// TIA Portal V18 export
FUNCTION_BLOCK "AndonMain"   // FB1, FBD
{ S7_Optimized_Access := 'TRUE' }
VERSION : 0.1
// stored: AutoNumber true, IsIECCheckEnabled false, IsRetainMemResEnabled false, MemoryReserve 100, SetENOAutomatically false, UDAEnableTagReadback false
   VAR
      fpBit_greenTrigger : Bool;
      AndonBoxASi_v2_Instance_8 { S7_SetPoint := 'True'} : "AndonBoxASi";
      AndonBoxASi_v2_Instance_9 { S7_SetPoint := 'True'} : "AndonBoxASi";
      AndonBoxASi_v2_Instance1 { S7_SetPoint := 'True'} : "AndonBoxASi";
      AndonBoxASi_v2_Instance2 { S7_SetPoint := 'True'} : "AndonBoxASi";
      AndonBoxASi_v2_Instance3 { S7_SetPoint := 'True'} : "AndonBoxASi";
      AndonBoxASi_v2_Instance4 { S7_SetPoint := 'True'} : "AndonBoxASi";
      AndonBoxASi_v2_Instance5 { S7_SetPoint := 'True'} : "AndonBoxASi";
      AndonBoxASi_v2_Instance6 { S7_SetPoint := 'True'} : "AndonBoxASi";
      AndonBoxASi_v2_Instance7 { S7_SetPoint := 'True'} : "AndonBoxASi";
      AndonBoxASi_v2_Instance10 { S7_SetPoint := 'True'} : "AndonBoxASi";
   END_VAR
   VAR_TEMP   // added for the SCL form of the ladder/FBD networks
      _w1 : Bool;
      _w2 : Bool;
   END_VAR
BEGIN

REGION Network 1: Green trigger
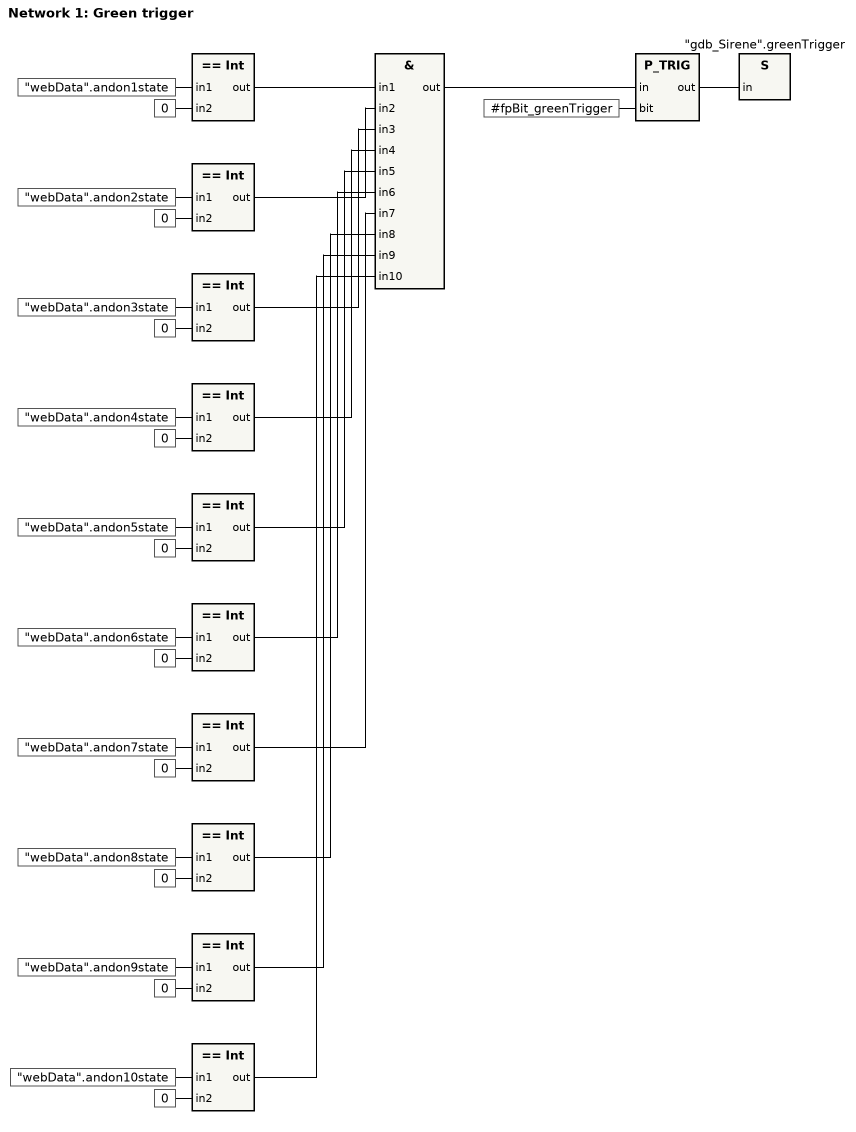
   #_w1 := ("webData".andon1state = 0) AND ("webData".andon2state = 0) AND ("webData".andon3state = 0) AND ("webData".andon4state = 0) AND ("webData".andon5state = 0) AND ("webData".andon6state = 0) AND ("webData".andon7state = 0) AND ("webData".andon8state = 0) AND ("webData".andon9state = 0) AND ("webData".andon10state = 0);
   #_w2 := #_w1 AND NOT #fpBit_greenTrigger;   // rising edge
   #fpBit_greenTrigger := #_w1;
   IF #_w2 THEN "gdb_Sirene".greenTrigger := TRUE; END_IF;
END_REGION

REGION Network 2: Andon1
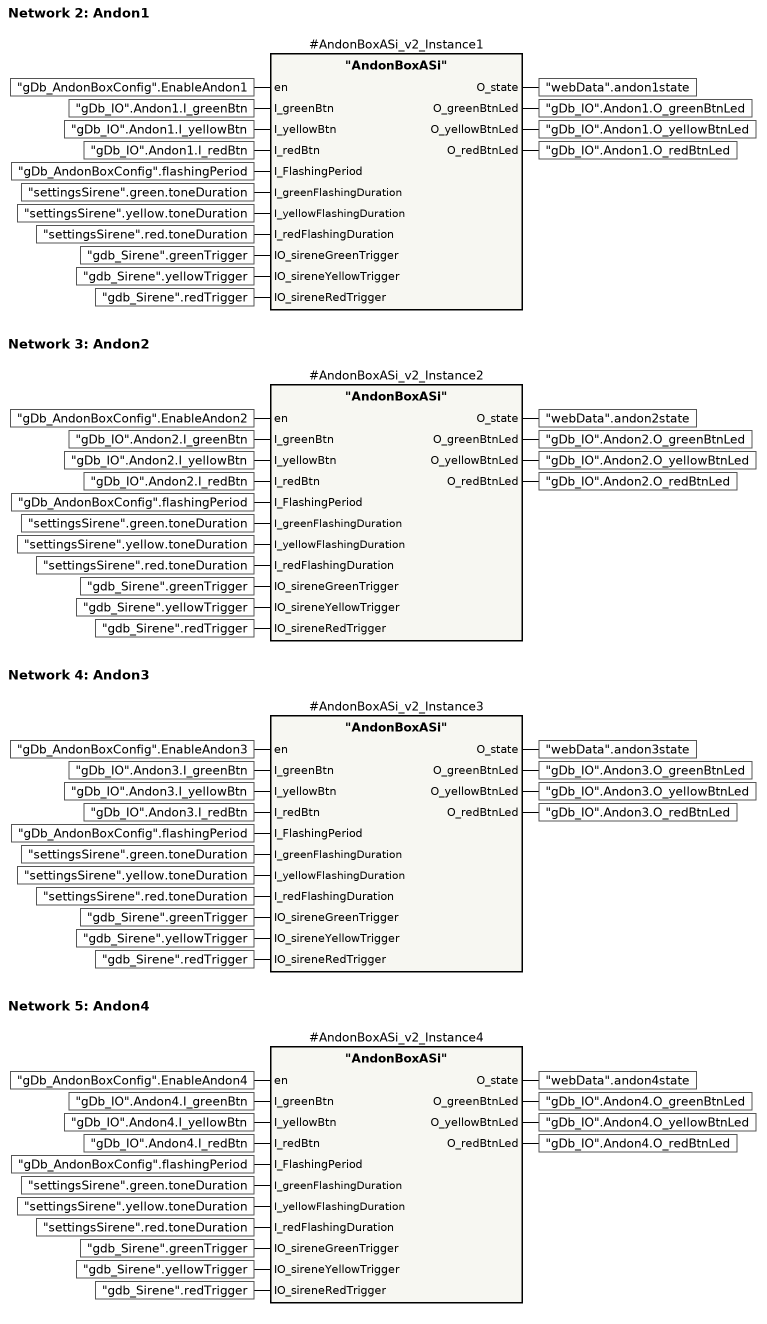
   IF "gDb_AndonBoxConfig".EnableAndon1 THEN
       #AndonBoxASi_v2_Instance1(I_greenBtn := "gDb_IO".Andon1.I_greenBtn,   // "AndonBoxASi"
                               I_yellowBtn := "gDb_IO".Andon1.I_yellowBtn,
                               I_redBtn := "gDb_IO".Andon1.I_redBtn,
                               I_FlashingPeriod := "gDb_AndonBoxConfig".flashingPeriod,
                               I_greenFlashingDuration := "settingsSirene".green.toneDuration,
                               I_yellowFlashingDuration := "settingsSirene".yellow.toneDuration,
                               I_redFlashingDuration := "settingsSirene".red.toneDuration,
                               IO_sireneGreenTrigger := "gdb_Sirene".greenTrigger,
                               IO_sireneYellowTrigger := "gdb_Sirene".yellowTrigger,
                               IO_sireneRedTrigger := "gdb_Sirene".redTrigger,
                               O_state => "webData".andon1state,
                               O_greenBtnLed => "gDb_IO".Andon1.O_greenBtnLed,
                               O_yellowBtnLed => "gDb_IO".Andon1.O_yellowBtnLed,
                               O_redBtnLed => "gDb_IO".Andon1.O_redBtnLed);
   END_IF;
END_REGION

REGION Network 3: Andon2
   IF "gDb_AndonBoxConfig".EnableAndon2 THEN
       #AndonBoxASi_v2_Instance2(I_greenBtn := "gDb_IO".Andon2.I_greenBtn,   // "AndonBoxASi"
                               I_yellowBtn := "gDb_IO".Andon2.I_yellowBtn,
                               I_redBtn := "gDb_IO".Andon2.I_redBtn,
                               I_FlashingPeriod := "gDb_AndonBoxConfig".flashingPeriod,
                               I_greenFlashingDuration := "settingsSirene".green.toneDuration,
                               I_yellowFlashingDuration := "settingsSirene".yellow.toneDuration,
                               I_redFlashingDuration := "settingsSirene".red.toneDuration,
                               IO_sireneGreenTrigger := "gdb_Sirene".greenTrigger,
                               IO_sireneYellowTrigger := "gdb_Sirene".yellowTrigger,
                               IO_sireneRedTrigger := "gdb_Sirene".redTrigger,
                               O_state => "webData".andon2state,
                               O_greenBtnLed => "gDb_IO".Andon2.O_greenBtnLed,
                               O_yellowBtnLed => "gDb_IO".Andon2.O_yellowBtnLed,
                               O_redBtnLed => "gDb_IO".Andon2.O_redBtnLed);
   END_IF;
END_REGION

REGION Network 4: Andon3
   IF "gDb_AndonBoxConfig".EnableAndon3 THEN
       #AndonBoxASi_v2_Instance3(I_greenBtn := "gDb_IO".Andon3.I_greenBtn,   // "AndonBoxASi"
                               I_yellowBtn := "gDb_IO".Andon3.I_yellowBtn,
                               I_redBtn := "gDb_IO".Andon3.I_redBtn,
                               I_FlashingPeriod := "gDb_AndonBoxConfig".flashingPeriod,
                               I_greenFlashingDuration := "settingsSirene".green.toneDuration,
                               I_yellowFlashingDuration := "settingsSirene".yellow.toneDuration,
                               I_redFlashingDuration := "settingsSirene".red.toneDuration,
                               IO_sireneGreenTrigger := "gdb_Sirene".greenTrigger,
                               IO_sireneYellowTrigger := "gdb_Sirene".yellowTrigger,
                               IO_sireneRedTrigger := "gdb_Sirene".redTrigger,
                               O_state => "webData".andon3state,
                               O_greenBtnLed => "gDb_IO".Andon3.O_greenBtnLed,
                               O_yellowBtnLed => "gDb_IO".Andon3.O_yellowBtnLed,
                               O_redBtnLed => "gDb_IO".Andon3.O_redBtnLed);
   END_IF;
END_REGION

REGION Network 5: Andon4
   IF "gDb_AndonBoxConfig".EnableAndon4 THEN
       #AndonBoxASi_v2_Instance4(I_greenBtn := "gDb_IO".Andon4.I_greenBtn,   // "AndonBoxASi"
                               I_yellowBtn := "gDb_IO".Andon4.I_yellowBtn,
                               I_redBtn := "gDb_IO".Andon4.I_redBtn,
                               I_FlashingPeriod := "gDb_AndonBoxConfig".flashingPeriod,
                               I_greenFlashingDuration := "settingsSirene".green.toneDuration,
                               I_yellowFlashingDuration := "settingsSirene".yellow.toneDuration,
                               I_redFlashingDuration := "settingsSirene".red.toneDuration,
                               IO_sireneGreenTrigger := "gdb_Sirene".greenTrigger,
                               IO_sireneYellowTrigger := "gdb_Sirene".yellowTrigger,
                               IO_sireneRedTrigger := "gdb_Sirene".redTrigger,
                               O_state => "webData".andon4state,
                               O_greenBtnLed => "gDb_IO".Andon4.O_greenBtnLed,
                               O_yellowBtnLed => "gDb_IO".Andon4.O_yellowBtnLed,
                               O_redBtnLed => "gDb_IO".Andon4.O_redBtnLed);
   END_IF;
END_REGION

REGION Network 6: Andon5
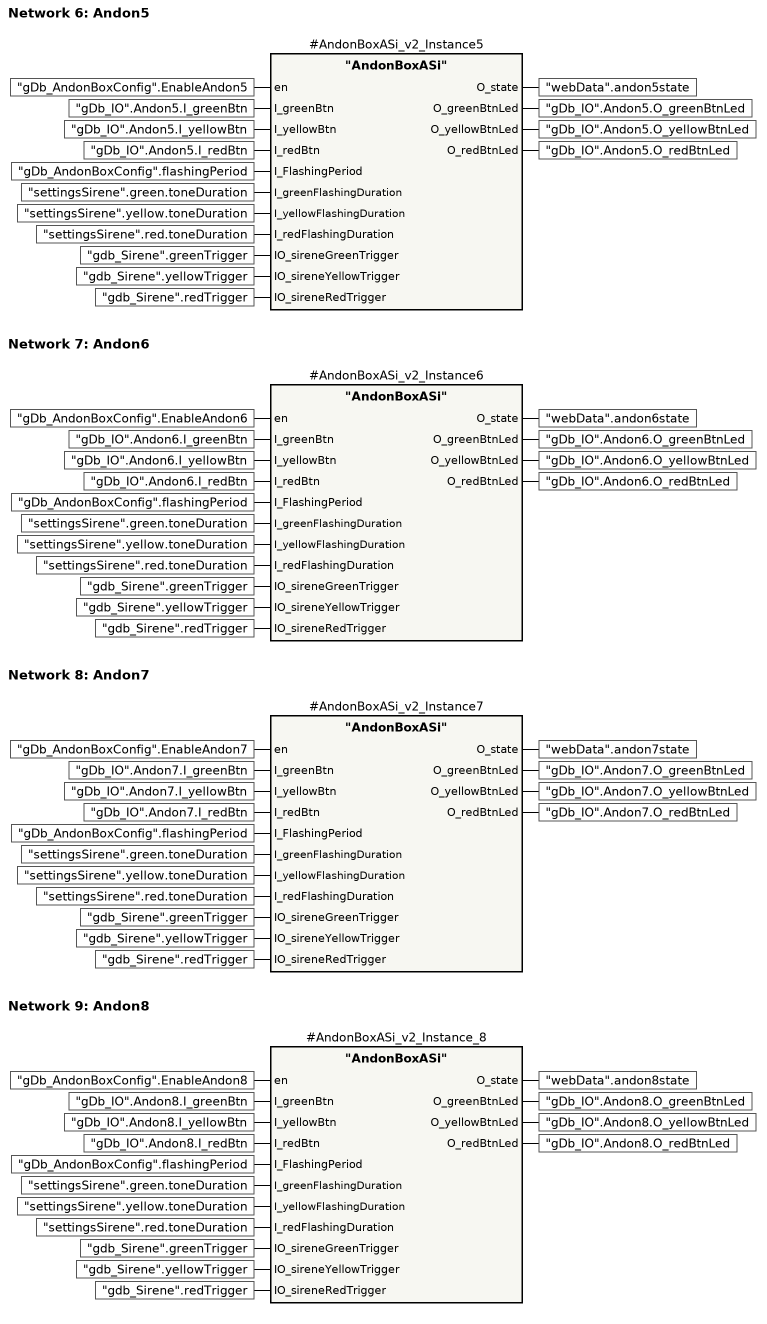
   IF "gDb_AndonBoxConfig".EnableAndon5 THEN
       #AndonBoxASi_v2_Instance5(I_greenBtn := "gDb_IO".Andon5.I_greenBtn,   // "AndonBoxASi"
                               I_yellowBtn := "gDb_IO".Andon5.I_yellowBtn,
                               I_redBtn := "gDb_IO".Andon5.I_redBtn,
                               I_FlashingPeriod := "gDb_AndonBoxConfig".flashingPeriod,
                               I_greenFlashingDuration := "settingsSirene".green.toneDuration,
                               I_yellowFlashingDuration := "settingsSirene".yellow.toneDuration,
                               I_redFlashingDuration := "settingsSirene".red.toneDuration,
                               IO_sireneGreenTrigger := "gdb_Sirene".greenTrigger,
                               IO_sireneYellowTrigger := "gdb_Sirene".yellowTrigger,
                               IO_sireneRedTrigger := "gdb_Sirene".redTrigger,
                               O_state => "webData".andon5state,
                               O_greenBtnLed => "gDb_IO".Andon5.O_greenBtnLed,
                               O_yellowBtnLed => "gDb_IO".Andon5.O_yellowBtnLed,
                               O_redBtnLed => "gDb_IO".Andon5.O_redBtnLed);
   END_IF;
END_REGION

REGION Network 7: Andon6
   IF "gDb_AndonBoxConfig".EnableAndon6 THEN
       #AndonBoxASi_v2_Instance6(I_greenBtn := "gDb_IO".Andon6.I_greenBtn,   // "AndonBoxASi"
                               I_yellowBtn := "gDb_IO".Andon6.I_yellowBtn,
                               I_redBtn := "gDb_IO".Andon6.I_redBtn,
                               I_FlashingPeriod := "gDb_AndonBoxConfig".flashingPeriod,
                               I_greenFlashingDuration := "settingsSirene".green.toneDuration,
                               I_yellowFlashingDuration := "settingsSirene".yellow.toneDuration,
                               I_redFlashingDuration := "settingsSirene".red.toneDuration,
                               IO_sireneGreenTrigger := "gdb_Sirene".greenTrigger,
                               IO_sireneYellowTrigger := "gdb_Sirene".yellowTrigger,
                               IO_sireneRedTrigger := "gdb_Sirene".redTrigger,
                               O_state => "webData".andon6state,
                               O_greenBtnLed => "gDb_IO".Andon6.O_greenBtnLed,
                               O_yellowBtnLed => "gDb_IO".Andon6.O_yellowBtnLed,
                               O_redBtnLed => "gDb_IO".Andon6.O_redBtnLed);
   END_IF;
END_REGION

REGION Network 8: Andon7
   IF "gDb_AndonBoxConfig".EnableAndon7 THEN
       #AndonBoxASi_v2_Instance7(I_greenBtn := "gDb_IO".Andon7.I_greenBtn,   // "AndonBoxASi"
                               I_yellowBtn := "gDb_IO".Andon7.I_yellowBtn,
                               I_redBtn := "gDb_IO".Andon7.I_redBtn,
                               I_FlashingPeriod := "gDb_AndonBoxConfig".flashingPeriod,
                               I_greenFlashingDuration := "settingsSirene".green.toneDuration,
                               I_yellowFlashingDuration := "settingsSirene".yellow.toneDuration,
                               I_redFlashingDuration := "settingsSirene".red.toneDuration,
                               IO_sireneGreenTrigger := "gdb_Sirene".greenTrigger,
                               IO_sireneYellowTrigger := "gdb_Sirene".yellowTrigger,
                               IO_sireneRedTrigger := "gdb_Sirene".redTrigger,
                               O_state => "webData".andon7state,
                               O_greenBtnLed => "gDb_IO".Andon7.O_greenBtnLed,
                               O_yellowBtnLed => "gDb_IO".Andon7.O_yellowBtnLed,
                               O_redBtnLed => "gDb_IO".Andon7.O_redBtnLed);
   END_IF;
END_REGION

REGION Network 9: Andon8
   IF "gDb_AndonBoxConfig".EnableAndon8 THEN
       #AndonBoxASi_v2_Instance_8(I_greenBtn := "gDb_IO".Andon8.I_greenBtn,   // "AndonBoxASi"
                               I_yellowBtn := "gDb_IO".Andon8.I_yellowBtn,
                               I_redBtn := "gDb_IO".Andon8.I_redBtn,
                               I_FlashingPeriod := "gDb_AndonBoxConfig".flashingPeriod,
                               I_greenFlashingDuration := "settingsSirene".green.toneDuration,
                               I_yellowFlashingDuration := "settingsSirene".yellow.toneDuration,
                               I_redFlashingDuration := "settingsSirene".red.toneDuration,
                               IO_sireneGreenTrigger := "gdb_Sirene".greenTrigger,
                               IO_sireneYellowTrigger := "gdb_Sirene".yellowTrigger,
                               IO_sireneRedTrigger := "gdb_Sirene".redTrigger,
                               O_state => "webData".andon8state,
                               O_greenBtnLed => "gDb_IO".Andon8.O_greenBtnLed,
                               O_yellowBtnLed => "gDb_IO".Andon8.O_yellowBtnLed,
                               O_redBtnLed => "gDb_IO".Andon8.O_redBtnLed);
   END_IF;
END_REGION

REGION Network 10: Andon9
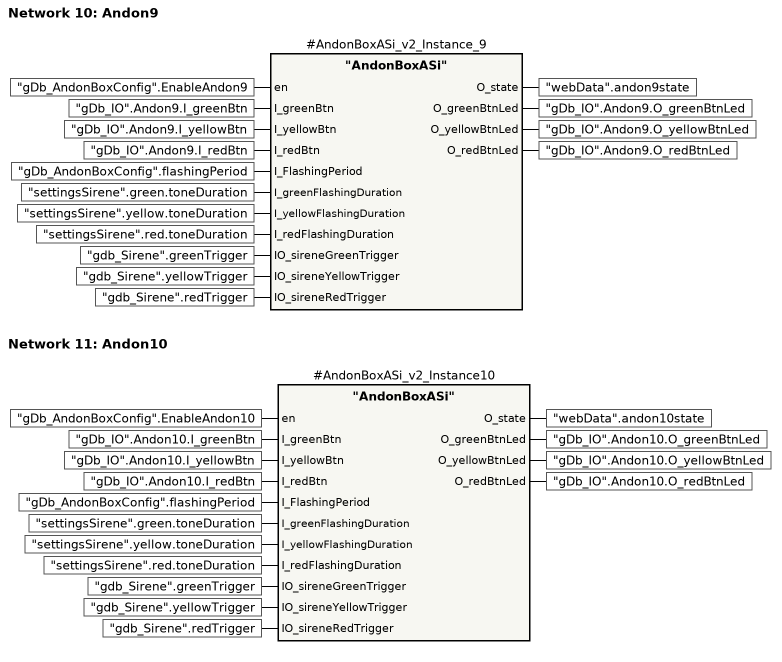
   IF "gDb_AndonBoxConfig".EnableAndon9 THEN
       #AndonBoxASi_v2_Instance_9(I_greenBtn := "gDb_IO".Andon9.I_greenBtn,   // "AndonBoxASi"
                               I_yellowBtn := "gDb_IO".Andon9.I_yellowBtn,
                               I_redBtn := "gDb_IO".Andon9.I_redBtn,
                               I_FlashingPeriod := "gDb_AndonBoxConfig".flashingPeriod,
                               I_greenFlashingDuration := "settingsSirene".green.toneDuration,
                               I_yellowFlashingDuration := "settingsSirene".yellow.toneDuration,
                               I_redFlashingDuration := "settingsSirene".red.toneDuration,
                               IO_sireneGreenTrigger := "gdb_Sirene".greenTrigger,
                               IO_sireneYellowTrigger := "gdb_Sirene".yellowTrigger,
                               IO_sireneRedTrigger := "gdb_Sirene".redTrigger,
                               O_state => "webData".andon9state,
                               O_greenBtnLed => "gDb_IO".Andon9.O_greenBtnLed,
                               O_yellowBtnLed => "gDb_IO".Andon9.O_yellowBtnLed,
                               O_redBtnLed => "gDb_IO".Andon9.O_redBtnLed);
   END_IF;
END_REGION

REGION Network 11: Andon10
   IF "gDb_AndonBoxConfig".EnableAndon10 THEN
       #AndonBoxASi_v2_Instance10(I_greenBtn := "gDb_IO".Andon10.I_greenBtn,   // "AndonBoxASi"
                               I_yellowBtn := "gDb_IO".Andon10.I_yellowBtn,
                               I_redBtn := "gDb_IO".Andon10.I_redBtn,
                               I_FlashingPeriod := "gDb_AndonBoxConfig".flashingPeriod,
                               I_greenFlashingDuration := "settingsSirene".green.toneDuration,
                               I_yellowFlashingDuration := "settingsSirene".yellow.toneDuration,
                               I_redFlashingDuration := "settingsSirene".red.toneDuration,
                               IO_sireneGreenTrigger := "gdb_Sirene".greenTrigger,
                               IO_sireneYellowTrigger := "gdb_Sirene".yellowTrigger,
                               IO_sireneRedTrigger := "gdb_Sirene".redTrigger,
                               O_state => "webData".andon10state,
                               O_greenBtnLed => "gDb_IO".Andon10.O_greenBtnLed,
                               O_yellowBtnLed => "gDb_IO".Andon10.O_yellowBtnLed,
                               O_redBtnLed => "gDb_IO".Andon10.O_redBtnLed);
   END_IF;
END_REGION

REGION Network 12: Semafor red
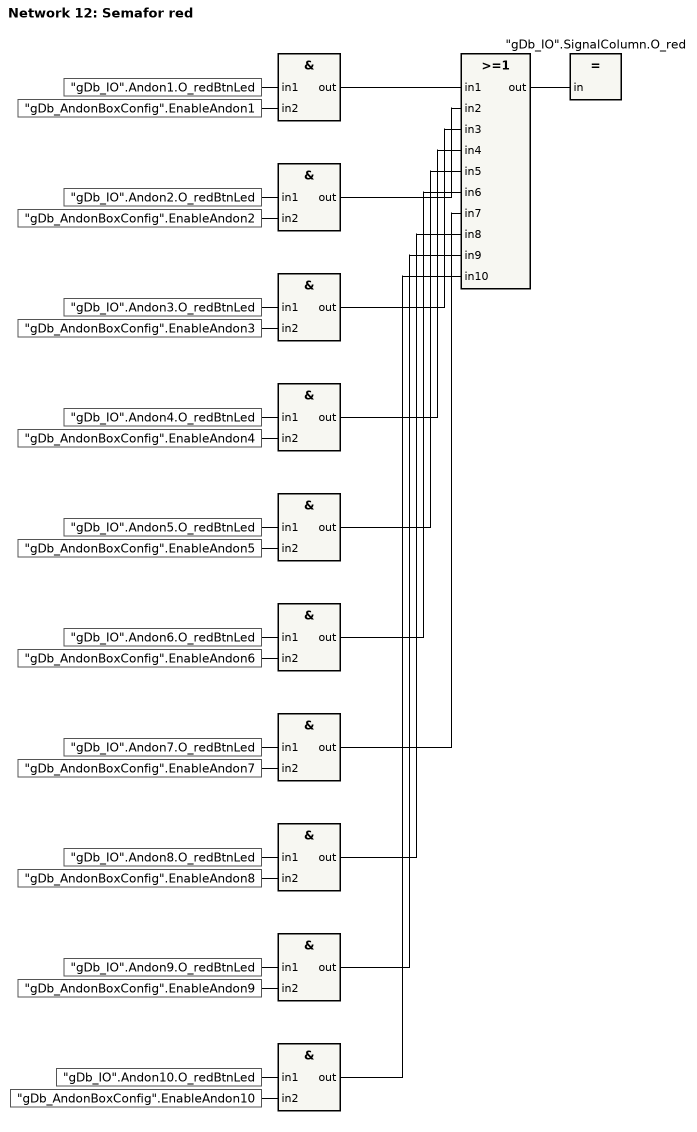
   "gDb_IO".SignalColumn.O_red := ("gDb_IO".Andon1.O_redBtnLed AND "gDb_AndonBoxConfig".EnableAndon1) OR ("gDb_IO".Andon2.O_redBtnLed AND "gDb_AndonBoxConfig".EnableAndon2) OR ("gDb_IO".Andon3.O_redBtnLed AND "gDb_AndonBoxConfig".EnableAndon3) OR ("gDb_IO".Andon4.O_redBtnLed AND "gDb_AndonBoxConfig".EnableAndon4) OR ("gDb_IO".Andon5.O_redBtnLed AND "gDb_AndonBoxConfig".EnableAndon5) OR ("gDb_IO".Andon6.O_redBtnLed AND "gDb_AndonBoxConfig".EnableAndon6) OR ("gDb_IO".Andon7.O_redBtnLed AND "gDb_AndonBoxConfig".EnableAndon7) OR ("gDb_IO".Andon8.O_redBtnLed AND "gDb_AndonBoxConfig".EnableAndon8) OR ("gDb_IO".Andon9.O_redBtnLed AND "gDb_AndonBoxConfig".EnableAndon9) OR ("gDb_IO".Andon10.O_redBtnLed AND "gDb_AndonBoxConfig".EnableAndon10);
END_REGION

REGION Network 13: Semafor yellow
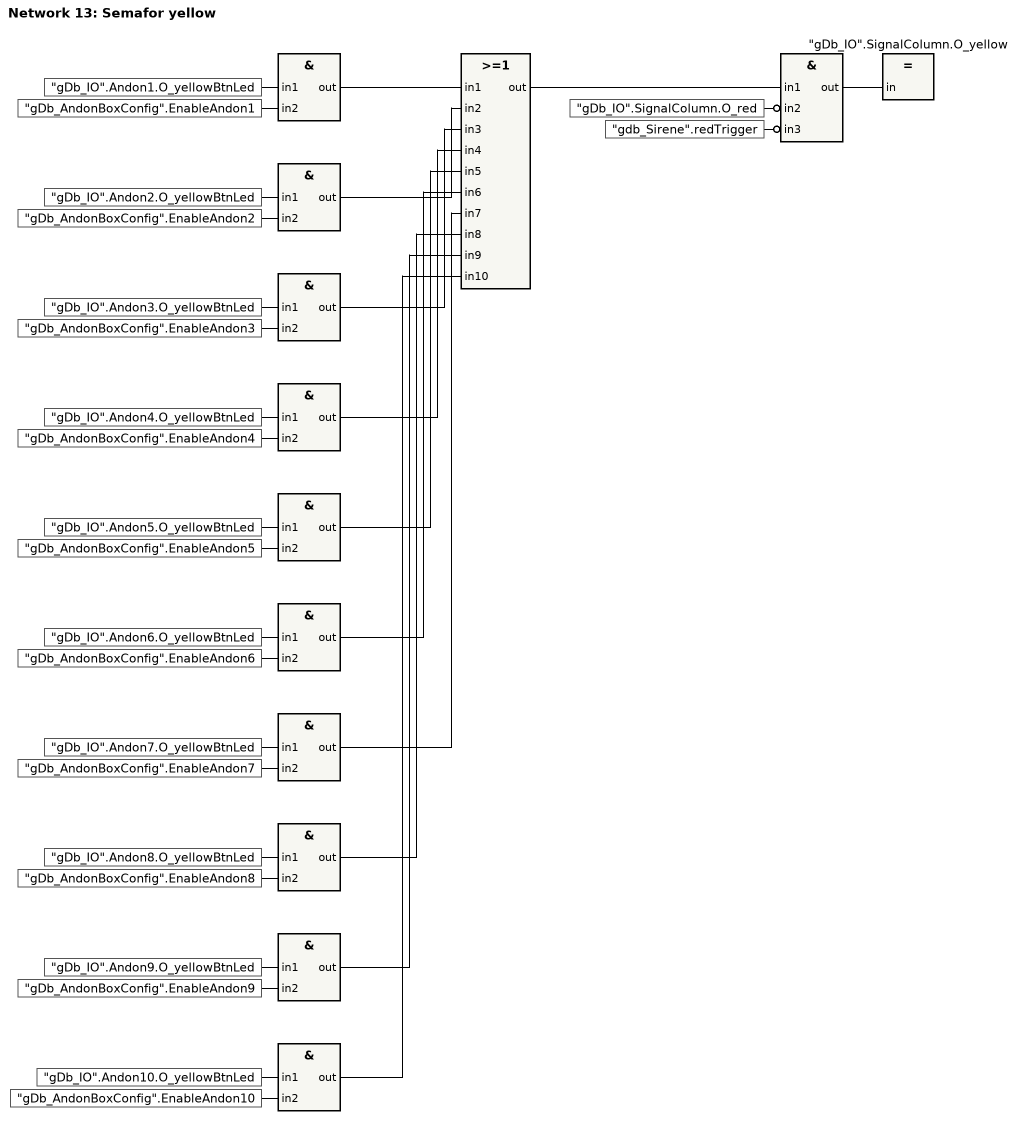
   "gDb_IO".SignalColumn.O_yellow := (("gDb_IO".Andon1.O_yellowBtnLed AND "gDb_AndonBoxConfig".EnableAndon1) OR ("gDb_IO".Andon2.O_yellowBtnLed AND "gDb_AndonBoxConfig".EnableAndon2) OR ("gDb_IO".Andon3.O_yellowBtnLed AND "gDb_AndonBoxConfig".EnableAndon3) OR ("gDb_IO".Andon4.O_yellowBtnLed AND "gDb_AndonBoxConfig".EnableAndon4) OR ("gDb_IO".Andon5.O_yellowBtnLed AND "gDb_AndonBoxConfig".EnableAndon5) OR ("gDb_IO".Andon6.O_yellowBtnLed AND "gDb_AndonBoxConfig".EnableAndon6) OR ("gDb_IO".Andon7.O_yellowBtnLed AND "gDb_AndonBoxConfig".EnableAndon7) OR ("gDb_IO".Andon8.O_yellowBtnLed AND "gDb_AndonBoxConfig".EnableAndon8) OR ("gDb_IO".Andon9.O_yellowBtnLed AND "gDb_AndonBoxConfig".EnableAndon9) OR ("gDb_IO".Andon10.O_yellowBtnLed AND "gDb_AndonBoxConfig".EnableAndon10)) AND NOT "gDb_IO".SignalColumn.O_red AND NOT "gdb_Sirene".redTrigger;
END_REGION

REGION Network 14: Semafor green
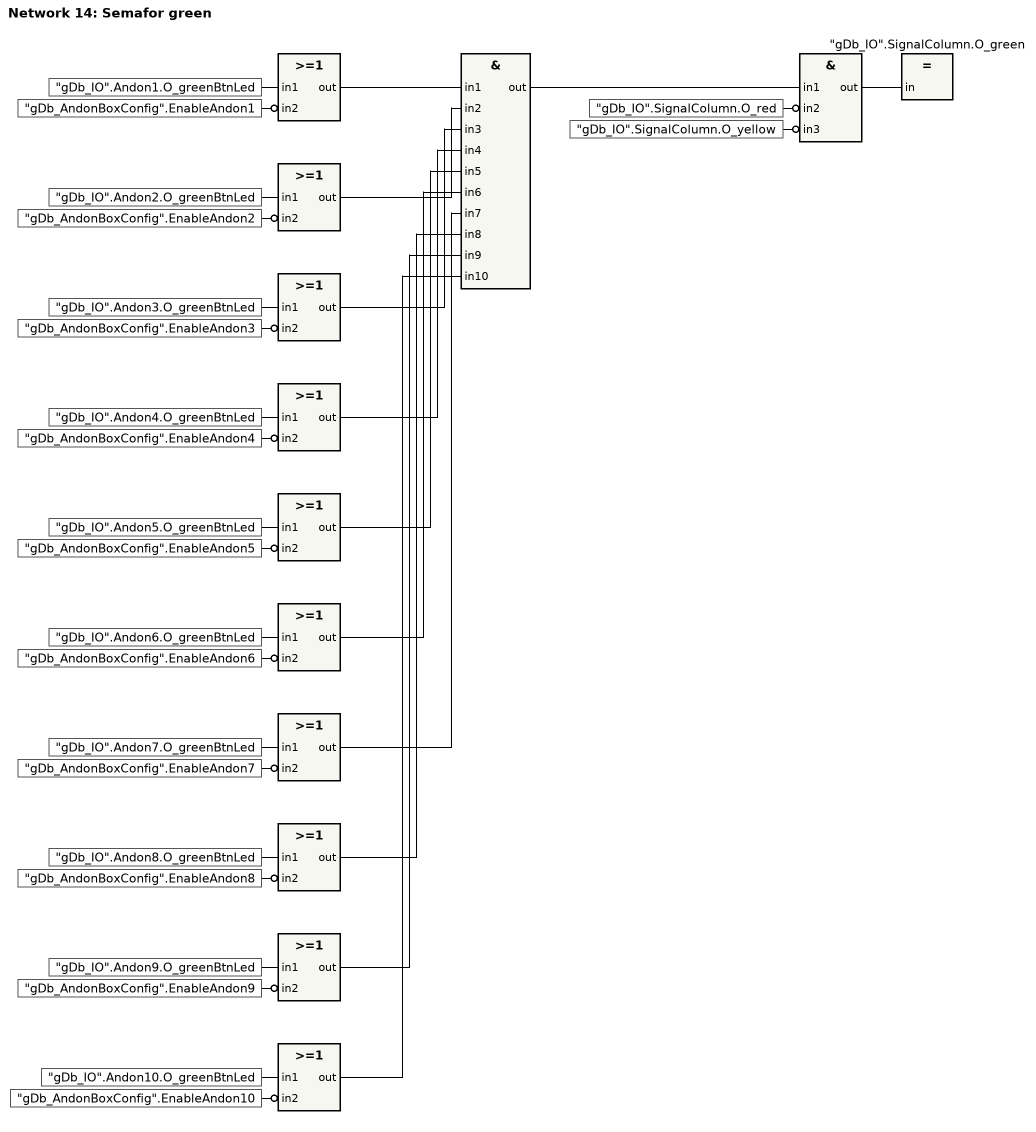
   "gDb_IO".SignalColumn.O_green := ("gDb_IO".Andon1.O_greenBtnLed OR NOT "gDb_AndonBoxConfig".EnableAndon1) AND ("gDb_IO".Andon2.O_greenBtnLed OR NOT "gDb_AndonBoxConfig".EnableAndon2) AND ("gDb_IO".Andon3.O_greenBtnLed OR NOT "gDb_AndonBoxConfig".EnableAndon3) AND ("gDb_IO".Andon4.O_greenBtnLed OR NOT "gDb_AndonBoxConfig".EnableAndon4) AND ("gDb_IO".Andon5.O_greenBtnLed OR NOT "gDb_AndonBoxConfig".EnableAndon5) AND ("gDb_IO".Andon6.O_greenBtnLed OR NOT "gDb_AndonBoxConfig".EnableAndon6) AND ("gDb_IO".Andon7.O_greenBtnLed OR NOT "gDb_AndonBoxConfig".EnableAndon7) AND ("gDb_IO".Andon8.O_greenBtnLed OR NOT "gDb_AndonBoxConfig".EnableAndon8) AND ("gDb_IO".Andon9.O_greenBtnLed OR NOT "gDb_AndonBoxConfig".EnableAndon9) AND ("gDb_IO".Andon10.O_greenBtnLed OR NOT "gDb_AndonBoxConfig".EnableAndon10) AND NOT "gDb_IO".SignalColumn.O_red AND NOT "gDb_IO".SignalColumn.O_yellow;
END_REGION
END_FUNCTION_BLOCK
